FUNCTION_BLOCK Ass_StackComv IMPLEMENTS ITF_AutoStructCommand
VAR_INPUT
END_VAR
VAR_OUTPUT
END_VAR
VAR
	strText	:STRING;
	i	:INT;
	_bProcessScan,_bInitialScan: BOOL;
	_bHalt , _bError,_bHaltPause: BOOL;
	nStep,nInitiStep  	: INT;
	_tmrT0,_tmrT1		:TON;
	bBoxPass: BOOL;
END_VAR

IF NOT _bInitialScan THEN
	nInitiStep	:= 0;
END_IF

_bInitialScan:=FALSE;



IF NOT _bProcessScan THEN
	nStep	:= 0;
END_IF

_bProcessScan:=FALSE;

{warning 'add property implementation'}
PROPERTY Connect : STRING(50)
GET
END_GET
SET
END_SET
END_PROPERTY

{warning 'add property implementation'}
PROPERTY Error : BOOL
GET
END_GET
END_PROPERTY

{warning 'add method implementation '}
METHOD ErrorClear : BOOL
END_METHOD

{warning 'add method implementation '}
METHOD FB_init : BOOL
VAR_INPUT
	(* if TRUE, the retain variables are initialized (warm start / cold start)*)
	bInitRetains	: BOOL;
	(* if TRUE, the instance afterwards gets moved into the copy code (online change)*)
	bInCopyCode	: BOOL;
END_VAR
END_METHOD

{warning 'add method implementation '}
METHOD HaltStepContiune : BOOL
END_METHOD

METHOD Initialization : BOOL
VAR_INPUT
	_Testmode	: BOOL;
END_VAR
_bInitialScan:=TRUE;

CASE nInitiStep OF
	0:		
		strText					:= 'ORG : Inital';
		Motor_Stack.qRun		:=FALSE;
		Vacm_StackUD			:=FALSE;
		Cyl_StackUD.qExtendCoil	:=FALSE;
		Bundling_yPause			:= FALSE;	
		nInitiStep				:= 5;	
	5:
		IF 	Cyl_StackUD.iOriginSensor THEN
			nInitiStep				:= 10;	
		END_IF;
	10:
			strText:='ORG : Done ';
			Initialization	:= TRUE;
	
END_CASE;
END_METHOD

{warning 'add property implementation'}
PROPERTY NoEntry : BOOL
GET
END_GET
END_PROPERTY

{warning 'add method implementation '}
METHOD Pause : BOOL
END_METHOD

METHOD Process : BOOL
VAR_INPUT
	bHlatMode	: BOOL;
END_VAR
_bProcessScan	:= TRUE;
CASE nStep OF 
	0:
		Vacm_StackUD			:=FALSE;
		Cyl_StackUD.qExtendCoil	:=FALSE;
		Motor_Stack.qRun		:=TRUE;
		nStep					:= 5;
		_tmrT0(IN:=FALSE);
		_tmrT1(IN:=FALSE);
	5:
		IF RunParameter.stack_bUsed THEN
				IF Sen_StackComvStop THEN
					Motor_Stack.qRun		:=FALSE;
					nStep					:= 9;
				END_IF
			ELSE		
		
			;
		
		
		END_IF
	9:
		_tmrT0(IN:=TRUE,PT:=T#1S);
		IF _tmrT0.Q THEN
			_tmrT0(IN:=FALSE);
			nStep					:= 10;
		END_IF		
		
	10://堆疊1
		Cyl_StackUD.qExtendCoil	:= TRUE;
		_tmrT0(IN:=TRUE,PT:=RunParameter.stack_DelayTime1);
		IF _tmrT0.Q THEN
			_tmrT0(IN:=FALSE);
			nStep					:= 15;
		END_IF
	15:
		Vacm_StackUD			:=TRUE;	
		_tmrT0(IN:=TRUE,PT:=T#1S);
		IF _tmrT0.Q THEN
			_tmrT0(IN:=FALSE);
			nStep					:= 20;
		END_IF
	20:
		Cyl_StackUD.qExtendCoil	:= FALSE;		
		IF Cyl_StackUD.iOriginSensor THEN
			nStep					:= 25;
		END_IF		
	25:
		Motor_Stack.qRun		:=TRUE;
		IF Sen_StackComvStop THEN
			Motor_Stack.qRun		:=FALSE;
			nStep					:= 30;
		END_IF	
	30:	
		_tmrT0(IN:=TRUE,PT:=T#1S);
		IF _tmrT0.Q THEN
			_tmrT0(IN:=FALSE);
			nStep					:= 35;
		END_IF		
	
	35:		
		Cyl_StackUD.qExtendCoil	:= TRUE;
		_tmrT0(IN:=TRUE,PT:=RunParameter.stack_DelayTime2);
		IF _tmrT0.Q THEN
			_tmrT0(IN:=FALSE);
			nStep					:= 40;
		END_IF		
	40:
		Cyl_StackUD.qExtendCoil	:= FALSE;
		Vacm_StackUD			:=FALSE;
		_tmrT0(IN:=TRUE,PT:=T#0.5S);
		IF _tmrT0.Q THEN
			_tmrT0(IN:=FALSE);
			nStep					:= 45;
		END_IF						
	45:
		Motor_Stack.qRun		:=TRUE;
		IF NOT Sen_StackComvStop THEN
			nStep					:=0;
		END_IF	
	
	
	
	
END_CASE
END_METHOD

{warning 'add property implementation'}
PROPERTY Status : STRING(50)
GET
END_GET
END_PROPERTY

END_FUNCTION_BLOCK

(* stored: Version 1.1.0.1, ProductVersion 3.1.4024.16
   POU Ass_StackComv: Id {4b25830c-f5af-4eac-9d4d-de80b24edd39}, SpecialFunc None
   Property Connect: Id {a371786e-bcec-4523-a384-a2bef8001a0c}
   Get Get: Id {c2b60847-59a1-4f2e-a761-a78ee112decd}
   Set Set: Id {0808dff4-5621-418e-a295-4266bc39503a}
   Property Error: Id {8e1996c5-689e-41dc-8771-ce949e06e94e}
   Get Get: Id {065378a1-67cf-4878-b432-41d5f2355425}
   Method ErrorClear: Id {a339a88e-b35e-48af-af47-02390217588e}
   Method FB_init: Id {95a8debb-1c67-4616-b911-0721a93f46e6}
   Method HaltStepContiune: Id {0dc00c82-e09c-4ec0-b9a3-23ac9ba5992d}
   Method Initialization: Id {68df2561-95fa-4481-b660-382046a2754b}
   Property NoEntry: Id {c2ac9021-b8c3-4fdc-8125-d256457068d6}
   Get Get: Id {f57af2ab-2034-46ea-af7f-472d3b7a0aa4}
   Method Pause: Id {7c2282fa-2483-4aff-a09f-26d3f1a27dc3}
   Method Process: Id {6448f121-61fb-4edd-a9d3-84894ee57953}
   Property Status: Id {b2ad1aac-7177-4ef5-aea5-5718cbec52b8}
   Get Get: Id {28a7eb0f-71f1-4cfc-85ef-c023d9fa3489} *)
